SUBAPPLICATION mapping_Uebung_012c (* String Input und Speichern (WIP) *)
  (* Standard: 61499-2; Description: Copyright (c) 2023 Meisterschulen am Ostbahnhof This program and the accompanying materials are made available under the terms of the Eclipse Public License 2.0 which is available at https://www.eclipse.org/legal/epl-2.0/ SPDX-License-Identifier: EPL-2.0 *)
  (* Version 1.0, 2023-10-23, Franz Höpfinger, Meisterschulen am Ostbahnhof *)
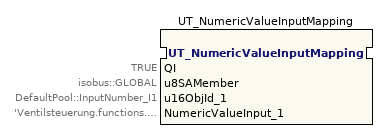
  FBS
    UT_NumericValueInputMapping : UT_NumericValueInputMapping(QI := TRUE, u8SAMember := isobus::GLOBAL, u16ObjId_1 := DefaultPool::InputNumber_I1, NumericValueInput_1 := 'Ventilsteuerung.functions.InputNumber_I1');
  END_FBS
END_SUBAPPLICATION
